Staubli VAL3: setPrd.pgx

program setPrd(string& x_sInOut[], string& x_sOut)
  local string l_sItemName
begin
  //
  x_sOut=""
  call PublicProg:addListItem(l_sItemName,x_sInOut,"P")
  if l_sItemName!=""
    //建立
    if x_sInOut[0]!=""
      insert(x_sInOut[size(x_sInOut)])
    endIf
    x_sInOut[size(x_sInOut)-1]=l_sItemName
    x_sOut=l_sItemName
    call user:listadd(l_sItemName)
  endIf
end
